// Base interface for an object.
INTERFACE I_Object EXTENDS __SYSTEM.IQueryInterface

END_INTERFACE

(* stored: Version 1.1.0.1, ProductVersion 3.1.4024.12
   Itf I_Object: Id {bd90aed1-a233-48b1-b5f3-285ade7adafd} *)
